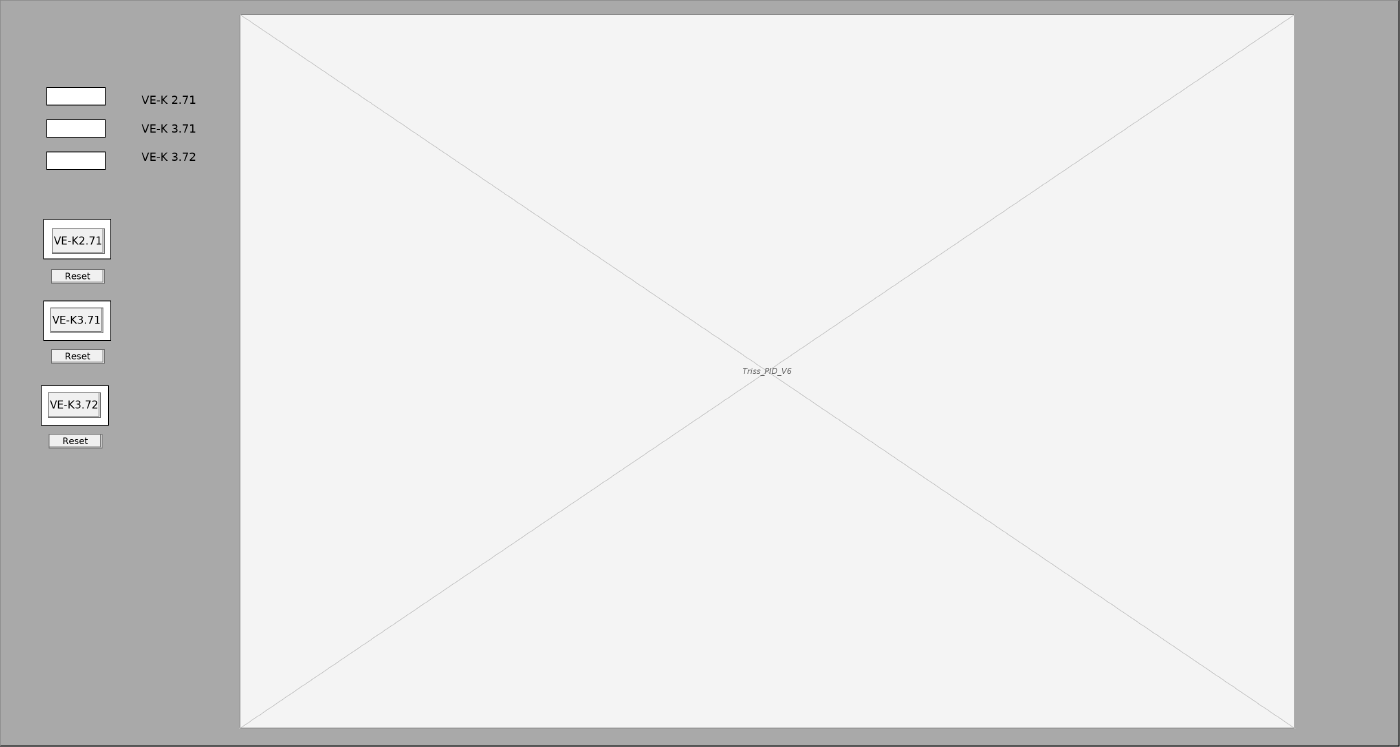
VISUALIZATION PID  // 1782x952, background image 
    Rectangle (0,950 1780x2)
    Rectangle (1780,0 2x950)
    Rectangle (55,279 86x51), colour toggle: GVL.V_Dampf_nach_Komp
    Button (66,291 67x32), "VE-K2.71"
        tap GVL.V_Dampf_nach_Komp_manu
    Button (65,343 68x18), "Reset"
        tap GVL.V_Dampf_nach_Komp_Reset
    Rectangle (55,383 86x51), colour toggle: V_Entlueftung_1
    Button (64,392 67x32), "VE-K3.71"
        tap V_Entlueftung_1_manu
    Button (65,445 68x18), "Reset"
        tap V_Entlueftung_1_Reset
    Rectangle (59,111 75x23), colour toggle: GVL.V_Dampf_nach_Komp_negiert
    Rectangle (59,152 75x23), colour toggle: V_Entlueftung_1_negiert
    Rectangle (143,86 144x156), "VE-K 2.71 VE-K 3.71 VE-K 3.72"
    Rectangle (52,491 86x51), colour toggle: V_Entlueftung_2
    Button (61,500 67x32), "VE-K3.72"
        tap V_Entlueftung_2_manu
    Button (62,553 68x18), "Reset"
        tap GVL.V_Entlueftung_2_Reset
    Rectangle (59,193 75x23), colour toggle: V_Entlueftung_2_negiert
    Image (305,18 1343x910), image: Triss_PID_V6
END_VISUALIZATION

(* stored: Version 1.1.0.1, ProductVersion 3.1.4024.3
   Visu PID: Id {07e37b6f-cf09-4b9c-afde-fc951a8e4364} *)
